PROGRAM MAIN
VAR
	alarms  : FB_AlarmHandler;
	
	// Start digin digout van appeltjes
	digIn_V2012_1 : FB_SimulatedDigIn;
	digIn_V2012_2 : FB_SimulatedDigIn;
	digOut_V2012 : FB_SimulatedDigOut;
	
	digIn_V2021_1 : FB_SimulatedDigIn;
	digIn_V2021_2 : FB_SimulatedDigIn;
	digOut_V2021 : FB_SimulatedDigOut;
	
	digIn_V2023_1 : FB_SimulatedDigIn;
	digIn_V2023_2 : FB_SimulatedDigIn;
	digOut_V2023 : FB_SimulatedDigOut;
	
	digIn_V2024_1 : FB_SimulatedDigIn;
	digIn_V2024_2 : FB_SimulatedDigIn;
	digOut_V2024 : FB_SimulatedDigOut;
	// Einde digin digout van appeltjes
	
	// Start digin digout van AFO
	digOutOpeningV2013 : FB_SimulatedDigOutOpen_AFO;
	digOutClosingV2013 :FB_SimulatedDigOutClose_AFO;
	AnaInV2013 : FB_SimulatedAnaIn_AFO;
	
	digOutOpeningV2022 : FB_SimulatedDigOutOpen_AFO;
	digOutClosingV2022 :FB_SimulatedDigOutClose_AFO;
	AnaInV2022 : FB_SimulatedAnaIn_AFO;
	// Einde digin digout van AFO

	V2012 : FB_OpenDichtKlep(tag := 'V2012', DigInClosed := digIn_V2012_1, DigInOpened := digIn_V2012_2, DigOut := digOut_V2012);
	V2021 : FB_OpenDichtKlep(tag := 'V2021', DigInClosed := digIn_V2021_1, DigInOpened := digIn_V2021_2, DigOut := digOut_V2021);
	V2023 : FB_OpenDichtKlep(tag := 'V2023', DigInClosed := digIn_V2023_1, DigInOpened := digIn_V2023_2, DigOut := digOut_V2023);
	V2024 : FB_OpenDichtKlep(tag := 'V2024', DigInClosed := digIn_V2024_1, DigInOpened := digIn_V2024_2, DigOut := digOut_V2024);  
	
	V2013_AFO : FB_Regelschuif_AFO;
	V2022_AFO : FB_Regelschuif_AFO;
	
	V2013_DG : FB_Regelschuif_DG;
	V2022_DG : FB_Regelschuif_DG;
	
	P2011 : FB_Pomp;
	P2021 : FB_Pomp;
	
	Regelingen : FB_Regelingen;
	
	ControllerInmalen : FB_Inmalen(OpenDichtKlepV2012 := V2012,
								   OpenDichtKlepV2021 := V2021, 
								   OpenDichtKlepV2023 := V2023, 
								   OpenDichtKlepV2024 := V2024,
								   RegelschuifV2013_AFO := V2013_AFO,
								   RegelschuifV2022_AFO := V2022_AFO,
								   RegelschuifV2013_DG := V2013_DG,
								   RegelschuifV2022_DG := V2022_DG,
								   PompP2021 := P2021 );
								   
									   
END_VAR

//Start function regelingen AFO
Regelingen ();
//End function regelingen AFO

//start functions kleppen appeltjes
digIn_V2012_1();
digIn_V2012_2();
digOut_V2012();

digIn_V2021_1();
digIn_V2021_2();
digOut_V2021();

digIn_V2023_1();
digIn_V2023_2();
digOut_V2023();

digIn_V2024_1();
digIn_V2024_2();
digOut_V2024();

V2012();
V2021();
V2023();
V2024();
//End  function kleppen appeltjes

//Start function inmalen appeltjes
ControllerInmalen ();
//End function inmalen appeltjes

END_PROGRAM

(* stored: Version 1.1.0.1, ProductVersion 3.1.4026.8
   POU MAIN: Id {e75b5398-c694-4eee-851b-9c5873361745}, SpecialFunc None *)
